{attribute 'GeneratedUsingTerminal: EL1918-0000-0016'}
{attribute addProperty BoxType "EL1918-0000-0016"}
{attribute addProperty Id "FSOEAT %I*FSOE_8C3E79C621"}
{attribute addProperty CRC "2384937038"}
{attribute addProperty Size "21"}
TYPE FSoE_Inputs_8E27404E :
STRUCT
	{attribute addProperty Name "FSOE"}
	FSOE AT %I* : FSOE_8C3E79C6;
END_STRUCT
END_TYPE

(* stored: Version 1.2.0.0, ProductVersion 3.1.4024.9
   DUT FSoE_Inputs_8E27404E: Id {d8cde3e8-817c-4389-a80c-9951b8ff73ee} *)
